PROGRAM ERROR_CASE_STATEMENT
VAR
END_VAR

CASE MOBILEHOIST.MAINSTATE OF
	
(*NORMAL OPERATION*)

	0:
		
	IF MOBILEHOIST.LOWERED_PROPERLY THEN
		
		MOBILEHOIST.MAINPWR			:= TRUE;
	
	END_IF


	
	IF MOBILEHOIST.ESTOP_CONDITION OR MOBILEHOIST.IOERROR OR MOBILEHOIST.TEMP_SWITCH = FALSE THEN
		
		MOBILEHOIST.MAINSTATE := 1;
		
	END_IF
	
	IF MOBILEHOIST.LOWERED_IMPROPERLY THEN
		
		MOBILEHOIST.MAINSTATE := 2;
		
	END_IF
	
	IF MOBILEHOIST.RAISED_PROPERLY THEN
		
		MOBILEHOIST.MAINSTATE := 3;
		
	END_IF
	
(*E-STOP/EMERGENCY MODE*)

	1:
	
	MOBILEHOIST.MAGNETIC_BRAKE1 	:= FALSE;
	MOBILEHOIST.MAGNETIC_BRAKE2 	:= FALSE;
	MOBILEHOIST.MAINPWR				:= FALSE;
	
	IF MOBILEHOIST.ESTOP_CONDITION = FALSE AND MOBILEHOIST.IOERROR = FALSE AND MOBILEHOIST.TEMP_SWITCH = FALSE THEN
		
		MOBILEHOIST.MAINSTATE := 0;
		
	END_IF
	
(*IMPROPERLY LOWERED*)

	2:
	
	MOBILEHOIST.MAGNETIC_BRAKE1 	:= FALSE;
	MOBILEHOIST.MAGNETIC_BRAKE2 	:= FALSE;
	MOBILEHOIST.MAINPWR				:= FALSE;

	IF MOBILEHOIST.LOWERED_IMPROPERLY = FALSE THEN
		
		MOBILEHOIST.MAINSTATE := 0;
		
	END_IF
	
(*PROPERLY RAISED*)
	
	3:
	
	MOBILEHOIST.MAGNETIC_BRAKE1 	:= FALSE;
	MOBILEHOIST.MAGNETIC_BRAKE2 	:= FALSE;
	MOBILEHOIST.MAINPWR				:= FALSE;

	IF MOBILEHOIST.RAISED_PROPERLY = FALSE THEN
		
		MOBILEHOIST.MAINSTATE := 0;
		
	END_IF
	
END_CASE

END_PROGRAM

(* stored: Version 1.1.0.1, ProductVersion 3.1.4024.11
   POU ERROR_CASE_STATEMENT: Id {5aed32b3-574f-4dcf-9953-063583c93cff}, SpecialFunc None *)
